{attribute addProperty BoxType "EL6201-0000-0017"}
{attribute addProperty Id "Slave_20A_DO0BIT10.125153Slave_20A_DO1BIT10.125154Slave_20A_DO2BIT10.125155Slave_20A_DO3BIT10.125156Slave_20B_DO0BIT10.125157Slave_20B_DO1BIT10.125158Slave_20B_DO2BIT10.125159Slave_20B_DO3BIT10.125160"}
{attribute addProperty CRC "1651529783"}
{attribute addProperty SizeInBites "8"}
{attribute addProperty SizeInBytes "1"}
TYPE Slave_20_Outputs_62705837 :
STRUCT
	{attribute addProperty Name "Slave_20A_DO0"}
	Slave_20A_DO0 : BIT;
	{attribute addProperty Name "Slave_20A_DO1"}
	Slave_20A_DO1 : BIT;
	{attribute addProperty Name "Slave_20A_DO2"}
	Slave_20A_DO2 : BIT;
	{attribute addProperty Name "Slave_20A_DO3"}
	Slave_20A_DO3 : BIT;
	{attribute addProperty Name "Slave_20B_DO0"}
	Slave_20B_DO0 : BIT;
	{attribute addProperty Name "Slave_20B_DO1"}
	Slave_20B_DO1 : BIT;
	{attribute addProperty Name "Slave_20B_DO2"}
	Slave_20B_DO2 : BIT;
	{attribute addProperty Name "Slave_20B_DO3"}
	Slave_20B_DO3 : BIT;
END_STRUCT
END_TYPE

(* stored: Version 1.2.0.0, ProductVersion 3.1.4024.9
   DUT Slave_20_Outputs_62705837: Id {f20cdec8-8ef6-4aa4-87a0-0fdd91e2b95f} *)
